FUNCTION_BLOCK AnalogOutputParametersFB
VAR_INPUT
END_VAR
VAR_OUTPUT
END_VAR
VAR
END_VAR

METHOD Update : BOOL
VAR_INPUT
	AO: REFERENCE TO GreenMasterAO_Base;
	Parameters: REFERENCE TO GreenMasterBaseParameters;
	AOut: AnalogOutputParameters;
END_VAR
AO.F_QN1 := AOut.F_QN1;
AO.T_GQ1 := AOut.T_GQ1;
AO.F_GQ1 := AOut.F_GQ1;
AO.C_QN1 := AOut.C_QN1;
AO.H_QN1 := AOut.H_QN1;
END_METHOD

END_FUNCTION_BLOCK

(* stored: Version 1.1.0.1, ProductVersion 3.1.4024.6
   POU AnalogOutputParametersFB: Id {c88c46c9-ad36-4d2f-906f-fabfc21039b1}, SpecialFunc None
   Method Update: Id {31ec9ef0-ffad-4ab2-ba4f-287b0d7de1d0} *)
